{attribute 'GeneratedUsingTerminal: EP9128-0021-0019'}
{attribute addProperty BoxType "EP9128-0021-0019"}
{attribute addProperty Id "A_0016_EP9214_0023_0019EP9214_7560C65380A_0017_EP9214_0023_0020EP9214_7560C65380A_0018_EP9214_0023_0021EP9214_7560C65380A_0019_EP9214_0023_0022EP9214_7560C65380A_0020_EP9224_0023_0016EP9224_2E4B686C112A_0021_EP9224_0023_0017EP9224_2E4B686C112A_0024_EP9521_0020_0000A_0024_EP9521_0020_0000_1CEF36B829A_0022_EP9224_0037_0017A_0022_EP9224_0037_0017_CE2477782A_0013_EP9128_0021_0019_2_EP9128_1021EP9128_1FC0878B2A_0013_EP9128_0021_0019_3_EP9128_2021EP9128_1FC0878B2"}
{attribute addProperty CRC "233182630"}
{attribute addProperty Size "579"}
TYPE A_0013_EP9128_0021_0019_0DE615A6 EXTENDS EP9128_1FC0878B :
STRUCT
	{attribute addProperty Name "A_0016_EP9214_0023_0019"}
	A_0016_EP9214_0023_0019 : EP9214_7560C653;
	{attribute addProperty Name "A_0017_EP9214_0023_0020"}
	A_0017_EP9214_0023_0020 : EP9214_7560C653;
	{attribute addProperty Name "A_0018_EP9214_0023_0021"}
	A_0018_EP9214_0023_0021 : EP9214_7560C653;
	{attribute addProperty Name "A_0019_EP9214_0023_0022"}
	A_0019_EP9214_0023_0022 : EP9214_7560C653;
	{attribute addProperty Name "A_0020_EP9224_0023_0016"}
	A_0020_EP9224_0023_0016 : EP9224_2E4B686C;
	{attribute addProperty Name "A_0021_EP9224_0023_0017"}
	A_0021_EP9224_0023_0017 : EP9224_2E4B686C;
	{attribute addProperty Name "A_0024_EP9521_0020_0000"}
	A_0024_EP9521_0020_0000 : A_0024_EP9521_0020_0000_1CEF36B8;
	{attribute addProperty Name "A_0022_EP9224_0037_0017"}
	A_0022_EP9224_0037_0017 : A_0022_EP9224_0037_0017_CE247778;
	{attribute addProperty Name "A_0013_EP9128_0021_0019_2_EP9128_1021"}
	A_0013_EP9128_0021_0019_2_EP9128_1021 : EP9128_1FC0878B;
	{attribute addProperty Name "A_0013_EP9128_0021_0019_3_EP9128_2021"}
	A_0013_EP9128_0021_0019_3_EP9128_2021 : EP9128_1FC0878B;
END_STRUCT
END_TYPE

(* stored: Version 1.2.0.0, ProductVersion 3.1.4024.9
   DUT A_0013_EP9128_0021_0019_0DE615A6: Id {f0baf034-ba30-43bc-b086-6c53cbab3a11} *)
